Staubli VAL3: RemoteControl.dtx

num VERSION = 1
sio socket = {link=UdpSocket\RemoteControl}
pointRx BASE_POSITION = {x=50, y=50, z=300, shoulder=sfree, elbow=efree, wrist=wfree, fatherId=world[0]}
jointRx BASE_POSE = {j1=-4.75879959898819E-06, j2=-86.5939224981684, j3=136.317941524159, j4=3.68060849006858E-06, j5=40.2759589805294, j6=-2.91771227743379E-06}
num MAGIC_HEADER = 149
string TASK_NAMES{}
  [MotionWorker] = "motionWorker"
  [MotionReporter] = "motionReporter"
  [MotionSupervisor] = "motionSupervisor"
  [SocketHandler] = "socketHandler"
  [MovingReporter] = "movingReporter"
tool endEffector = {x=660, fatherId=mount[0]}
tool mount = {ry=-90, fatherId=flange[0]}
bool motionQueued
num motionType
num reportInterval
pointRx target = {shoulder=sfree, elbow=efree, wrist=wfree, fatherId=world[0]}
mdesc NOMINAL_CONFIG = {accel=25, decel=25, blend=off}
mdesc SLOW_CONFIG = {accel=25, decel=25, tmax=150, rmax=50, blend=off}
mdesc moveConfig = {blend=off}
jointRx pose
tool selectedTool = {fatherId=flange[0]}
bool reportEnabled
configRx ARM_CONFIG = {shoulder=sfree, elbow=efree, wrist=wfree}
pointRx intermediate = {fatherId=world[0]}
